//Load arbiter with beam parameter sets
AssertTrue(fbArbiter.AddRequest(nEVReqID, stEVReqBP, sDevName:= 'Device'),
                    'Safest stEVReqBP request failed to load');

//Load arbiter with beam parameter sets
AssertTrue(fbArbiter.AddRequest(nRateReqID, stRateReqBP, sDevName:= 'Device'),
                    'Safest stRateReqBP request failed to load');

//Load arbiter with beam parameter sets
AssertTrue(fbArbiter.AddRequest(nBCRangeReqID, stBCReqBP, sDevName:= 'Device'),
                    'Safest stBCReqBP request failed to load');

stArbitratedBP := fbArbiter.GetArbitratedBP();

AssertFalse(F_DifferentBeamParams(stExpectedBP, stArbitratedBP),
                'Arbitrated BP does not match expected.');

TEST_FINISHED();
END_METHOD

METHOD DoS
VAR



    nOrigReqID : UDINT := 30;
    nSecondReqID : UDINT := 35;

    nPeskyReqID : UDINT := 40;


END_VAR
VAR_INST
    DosArb : FB_Arbiter(20);

    DummyHA : FB_DummyHA := (ReqAcknowledged:=FALSE); // Set req ack false to start so we can control when it is verified
    nTimeoutCounter : UINT;
    bInit : BOOL;
    bSecond : BOOL;
    eDosTestCases : E_ArbDosTestStates;
END_VAR
VAR CONSTANT
        nTimeoutCounterMAX : UINT := 50;
        nWaitCount : UINT := 10;
        nWait2ndCount : UINT := nWaitCount + 5;
END_VAR
TEST('DoS');

CASE eDosTestCases OF
    E_ArbDosTestStates.Init: // Init, first request
        DosArb.AddRequest(nOrigReqID, PMPS_GVL.cst0RateBeam, sDevName:= 'Device');
        eDosTestCases := E_ArbDosTestStates.SecondReq;

    E_ArbDosTestStates.SecondReq: // Add second request
        DosArb.AddRequest(nSecondReqID, PMPS_GVL.cst0RateBeam, sDevName:= 'Device');
        eDosTestCases := E_ArbDosTestStates.WaitForAck;

    E_ArbDosTestStates.WaitForAck:
        IF nTimeoutCounter > nWaitCount THEN
            DummyHA.ReqAcknowledged := TRUE;
            eDosTestCases := E_ArbDosTestStates.WaitFor2ndAck;
        END_IF

    E_ArbDosTestStates.WaitFor2ndAck:
        DummyHA.ReqAcknowledged := False;
        IF nTimeoutCounter > nWait2ndCount THEN
            DummyHA.ReqAcknowledged := TRUE;
            eDosTestCases := E_ArbDosTestStates.RunAsserts;
        END_IF

END_CASE

DosArb.ElevateRequest(DummyHA);

// Pesky request always adding and removing
DosArb.RemoveRequest(nPeskyReqID);
DosArb.AddRequest(nPeskyReqID, PMPS_GVL.cst0RateBeam, sDevName:= 'Device');


nTimeoutCounter := nTimeoutCounter + 1;

IF nTimeoutCounter > nTimeoutCounterMAX or eDosTestCases = E_ArbDosTestStates.RunAsserts THEN
    AssertTrue(DosArb.CheckRequest(nOrigReqID), 'Original request still not accepted');
    AssertTrue(DosArb.CheckRequest(nSecondReqID), 'Second request still not accepted');

    TEST_FINISHED_NAMED('DoS');
END_IF
END_METHOD

{attribute 'no_check'}
METHOD FullArbitrationStack
VAR_INPUT
END_VAR
VAR
    nId    :    DWORD := 1;
    stReq    :    ST_BeamParams := (nTran:=12);

    nIdDoS : DWORD := 13;
    stDoSReq : ST_BeamParams := PMPS_GVL.cstFullBeam;
END_VAR
VAR_INST
    fbArbiter    :    FB_Arbiter(1);

    fbHigherArb : FB_Arbiter(2);

    fbSubSysToArb : FB_SubSysToArbiter_IO; // Subsystem interface with beamline arbiter PLC
    pBPR : POINTER TO ST_BeamParams_IO;

    fbArbToSubSys : FB_ArbiterToSubSys_IO := (RequestingSystemID:=42); // Beamline arbiter PLC interface with subsystems
    pBPC : POINTER TO ST_BeamParams_IO;

    fbBPR : FB_BPRequestor; // Use in the arbiter PLC to apply an arbitrated beam parameter set to the accelerator interface

    FFO : FB_HardwareFFOutput; // Dummy FFO not important for these tests

    Cycle : INT := 0;

    CycleLimit : INT := 20;

END_VAR
VAR CONSTANT
    SysID : DWORD := 42;
END_VAR
// This simulates a synchronous cycle between the subsystem and arbiter PLC cycles. Ie. phase is locked, and cycle time is the same. This is not always the case, so these tests should be
// trusted with a grain of salt.

TEST('FullStack');



CASE Cycle OF

0:
    IF NOT fbArbiter.CheckRequestInPool(nID) THEN
        AssertTrue(fbArbiter.AddRequest(nId, stReq,'Device'), 'Arbiter returned false from AddRequest'); // some device asking its local arbiter for some beam parameters
    END_IF

    TEST('JustEnteredRequest');
    AssertFalse(fbArbiter.CheckRequest(nId),
        'Check should fail. Request not arbitrated yet.');
    TEST_FINISHED();

8000:
    TEST_FINISHED_NAMED('FullStack');

END_CASE


TEST('VerifyBPRHasBP');
IF fbHigherArb.CheckRequest(SysID) THEN
    AssertFalse(F_DifferentBeamParams(stReq, fbBPR.q_ReqBP),
        'Beam parameters not fully propagated to BPR at highest level');
        TEST_FINISHED_NAMED('VerifyBPRHasBP');
END_IF

TEST('ArbToSubsysPropagation');
IF fbArbToSubSys.nActiveCohort = fbArbToSubSys.nRequestedCohort
    AND fbArbToSubSys.nActiveCohort <> 0 THEN
    AssertTrue(fbHigherArb.CheckRequest(SysID),
        'Active cohort = Requested cohort before higher arbiter confirmed request was active');
    TEST_FINISHED_NAMED('ArbToSubsysPropagation');
END_IF

TEST('SubsysToArbPropagation');
IF fbArbiter.CheckRequest(nId) THEN
    AssertTrue(fbSubSysToArb.nActiveCohort >= fbSubSysToArb.nRequestCohort,
        'Request validated before higher level confirmation');
    TEST_FINISHED_NAMED('SubsysToArbPropagation');
END_IF


TEST('VerifyIncludedAtAllLevels');
IF fbArbiter.CheckRequest(nId) THEN
    AssertTrue(fbHigherArb.CheckRequest(fbArbToSubSys.RequestingSystemID), 'HigherArb is not yet included in arbitration');
    AssertTrue(fbSubSysToArb.CheckRequest(fbArbiter.nLowerAuthorityID), 'Local Arb is not yet included in arbitration');
    TEST_FINISHED_NAMED('VerifyIncludedAtAllLevels');
END_IF


///////////////////////////////////////
//Sub system cycle
fbSubSysToArb(Arbiter := fbArbiter, fbFFHWO := FFO);
//END of sub system cycle
///////////////////////////////////////

//Ethercat transfer simulation
// Transfer of requested BP to arbiter PLC
pBPR := ADR(fbArbToSubSys.i_RequestedBP);
pBPR^ := fbSubSysToArb.q_stRequestedBP;

// Transfer of current BP to sub system PLC
pBPC := ADR(fbSubSysToArb.i_stCurrentBP);
pBPC^ := fbArbToSubSys.o_CurrentBP;

//////////////////////////////////////
//Start of arbiter plc cycle
//Arb io collects sub system status
fbArbToSubSys(Arbiter := fbHigherArb, fbFFHWO := FFO); // This is making a request in the higher arb
//BPR collects arbiter summation
fbBPR(Arbiter := fbHigherArb); // This is getting the arbitrated BP




IF CycleLimit > Cycle THEN
    Cycle := Cycle + 1;
ELSE
    Cycle := 8000;
END_IF
END_METHOD

METHOD RemoveReq
VAR

    Arb : FB_Arbiter(20);

    DummyHA : FB_DummyHA;

    Result : BOOL;

END_VAR

Arb.AddRequest(30, PMPS_GVL.cst0RateBeam, 'Device');

Arb.ElevateRequest(DummyHA);

TEST('Remove Req');
    Result := Arb.RemoveRequest(77);

    AssertFalse( Result, 'RemoveReq returned true, with nothing to remove');
    AssertFalse( Arb.bStartNewAckRequest , 'StartNewAckRequest is set. Something is wrong');

TEST_FINISHED();
END_METHOD

METHOD RequestCheckRemoveBP
VAR_INPUT
END_VAR
VAR

    nId    :    DWORD := 1;
    stReq    :    ST_BeamParams;
END_VAR
VAR_INST
    fbArbiter    :    FB_Arbiter(1);
END_VAR
TEST('RequestBP');
AssertTrue(fbArbiter.AddRequest(nId, stReq, 'Device'),
    'Request failed');

TEST_FINISHED();

TEST('DuplicateID');
AssertFalse(fbArbiter.AddRequest(nId, stReq, 'Device'),
    'Duplicate request accepted, not good.');

TEST_FINISHED();

TEST('CheckBP');
AssertFalse(fbArbiter.CheckRequest(nId),
    'Check should fail. Request not arbitrated yet.');
TEST_FINISHED();

TEST('CheckBPArbitrated');
WRITE_PROTECTED_ULINT(ADR(fbArbiter.nActiveCohort), fbArbiter.nNextCohort);
AssertTrue(fbArbiter.CheckRequest(nId),
    'Check should pass.');

TEST_FINISHED();

TEST('IDDoesNotExist');

AssertFalse(fbArbiter.CheckRequest(nId+1),
    'Check returned true when ID does not exist');

TEST_FINISHED();

TEST('RemoveBP');
AssertTrue(fbArbiter.RemoveRequest(nId),
    'Remove failed');
AssertFalse(fbArbiter.CheckRequest(nId),
    'Remove did not remove request');

TEST_FINISHED();

TEST('NoRequestsFullBeam');

AssertFalse(F_DifferentBeamParams(fbArbiter.GetArbitratedBP(), PMPS_GVL.cstFullBeam), 'Arbitrated beam should be full with all requests removed');

TEST_FINISHED();
END_METHOD

METHOD StackArbiters
VAR_INPUT
END_VAR
VAR
    nId    :    DWORD := 1;
    stReq    :    ST_BeamParams := (nTran:=12);
END_VAR
VAR_INST
    fbArbiter    :    FB_Arbiter(1);

    fbHigherArb : FB_Arbiter(2);

    ArbBP : ST_BeamParams;

    Cycle : INT := 0;

    CycleLimit : INT := 20;

END_VAR
VAR CONSTANT
    SysID : DWORD := 42;
END_VAR

TEST('StackingArbiters');
fbArbiter.AddRequest(nReqID:=nId, stReqBP:=stReq, sDevName :='Device');

fbArbiter.ElevateRequest(fbHigherArb);

ArbBP := fbHigherArb.GetArbitratedBP();

AssertTrue(ArbBP.nTran = 12, 'We should see the transmission number here');

TEST_FINISHED();
END_METHOD

END_FUNCTION_BLOCK

// TestComponents/FB_ArbToSubsys_Test
{attribute 'call_after_init'}
FUNCTION_BLOCK FB_ArbToSubsys_Test EXTENDS TcUnit.FB_TestSuite
VAR_INPUT
END_VAR
VAR_OUTPUT
END_VAR
VAR
END_VAR

BasicFunction();

{attribute 'no_check'}
METHOD BasicFunction
VAR_INPUT
END_VAR
VAR CONSTANT
    SysID : DWORD := 42;
END_VAR
VAR
    nId    :    DWORD := 1;
    stReq    :    ST_BeamParams := (nTran:=12);
END_VAR
VAR_INST
    fbArbiter    :    FB_Arbiter(1);

    pBPR : POINTER TO ST_BeamParams_IO;

    stBPRIO : ST_BeamParams_IO := (
        nCohortInt := 1,
        nTran := 35); // Simulates subsystem BP request

    fbArbToSubSys : FB_ArbiterToSubSys_IO := (RequestingSystemID:=42); // Beamline arbiter PLC interface with subsystems
    pBPC : POINTER TO ST_BeamParams_IO;

    fbBPR : FB_BPRequestor; // Use in the arbiter PLC to apply an arbitrated beam parameter set to the accelerator interface

    FFO : FB_HardwareFFOutput; // Dummy FFO not important for these tests

    Cycle : INT := 0;

    CycleLimit : INT := 20;

END_VAR

// Simulate an initial cycle with no new requests coming in
fbBPR(Arbiter:=fbArbiter);
fbArbToSubSys(Arbiter:=fbArbiter, fbFFHWO:=FFO);

TEST('Init');
TEST_FINISHED();

//Ethercat transfer simulation
// Transfer of requested BP to arbiter PLC
pBPR := ADR(fbArbToSubSys.i_RequestedBP);
pBPR^ := stBPRIO;

///////////////////////////////////////
//Sub system cycle
fbBPR(Arbiter:=fbArbiter);
fbArbToSubSys(Arbiter:=fbArbiter, fbFFHWO:=FFO);
//END of sub system cycle
///////////////////////////////////////


TEST('New request');
    AssertTrue(fbArbToSubSys.nRequestedCohort = fbArbToSubSys.i_RequestedBP.nCohortInt, 'ReqCohort and qBP Cohort do not match, and they should');
    AssertTrue(fbArbiter.CheckRequestInPool(SysID), 'ArbToSubSys request should be in arbiter pool now');
    AssertTrue(fbArbToSubSys.nActiveCohort = 0, 'Active cohort should remain the initial value until the current request is active in higher arbitration');
    AssertTrue(fbArbToSubSys.o_CurrentBP.nCohortInt = fbArbToSubSys.nActiveCohort, 'Cohort being sent to sub system remains unincremented');
TEST_FINISHED_NAMED('New request');


///////////////////////////////////////
//Sub system cycle
fbBPR(Arbiter:=fbArbiter);
fbArbToSubSys(Arbiter:=fbArbiter, fbFFHWO:=FFO);
//END of sub system cycle
///////////////////////////////////////

///////////////////////////////////////
//Sub system cycle
fbBPR(Arbiter:=fbArbiter);
fbArbToSubSys(Arbiter:=fbArbiter, fbFFHWO:=FFO);
//END of sub system cycle
///////////////////////////////////////

///////////////////////////////////////
//Sub system cycle
fbBPR(Arbiter:=fbArbiter);
fbArbToSubSys(Arbiter:=fbArbiter, fbFFHWO:=FFO);
//END of sub system cycle
///////////////////////////////////////

TEST('Request has become active');
    AssertTrue(fbArbToSubSys.nRequestedCohort = fbArbToSubSys.nActiveCohort, 'ReqCohort and qBP Cohort do not match, and they should');
    AssertTrue(fbArbiter.CheckRequest(SysID), 'ArbToSubSys request should be in arbiter pool now');
    AssertTrue(fbArbToSubSys.nActiveCohort = stBPRIO.nCohortInt, 'Active cohort should remain the initial value until the current request is active in higher arbitration');
    AssertTrue(fbBPR.q_ReqBP.nTran = stBPRIO.nTran, 'BPR and requested BP should match');
TEST_FINISHED_NAMED('Request has become active');
END_METHOD

END_FUNCTION_BLOCK

// TestComponents/FB_AttenuatorSimulator
FUNCTION_BLOCK FB_AttenuatorSimulator
VAR_INPUT
    i_rRequestedAttenuation    :    REAL;
    i_stBPReadback    :    ST_BeamParams;
END_VAR
VAR_OUTPUT
    q_xFault    :    BOOL;
    q_rCurrentAttenuation    :    REAL;
END_VAR
VAR_IN_OUT
    Arbiter    :    FB_Arbiter; //Higher level arbiter from which upstream attenuation can be requested
END_VAR
VAR
    tonDelay    :    TON := (
        PT := T#3S
        );
END_VAR

// Really basic delay
tonDelay(IN := i_rRequestedAttenuation <> q_rCurrentAttenuation);

IF tonDelay.Q THEN
    q_rCurrentAttenuation := i_rRequestedAttenuation;
END_IF

END_FUNCTION_BLOCK

// TestComponents/FB_BPTM_Test
{attribute 'call_after_init'}
FUNCTION_BLOCK FB_BPTM_Test EXTENDS TcUnit.FB_TestSuite
VAR_INPUT
END_VAR
VAR_OUTPUT
END_VAR
VAR
END_VAR
VAR CONSTANT
    BPTM_ARR : UDINT := PMPS_PARAM.MAX_ASSERTIONS;
    cCycle : UINT := 20; // How many cycles does it take to complete a BPTM
END_VAR

BPTMBasicFunction();
InterruptAtAllSteps();
FullArbError();

METHOD BPTMBasicFunction
VAR_INPUT
END_VAR
VAR
    //Final and transition assertions
    nTransitionID    :    UDINT := 1;
    stTransitionAssertion    :    ST_BeamParams := (nRate := 10, nBCRange:=0);

    nReqID    :    UDINT    := 2;
    stReqAssertion    :    ST_BeamParams := (nTran := 0.2, nBCRange:=2#0000_0000_0000_0011);

END_VAR
VAR_INST
    fbBPTM_TestBasicFunction    :    BeamParameterTransitionManager;
    fbArbiter    :    FB_Arbiter(1);
    ffo : FB_HardwareFFOutput;
    fbSubSysIO : FB_DummyArbIO;
    xFirstPass    :    BOOL := TRUE;
    eTestStep: E_BPTMTestStates := E_BPTMTestStates.Init;
END_VAR

// Completes arbiter request elevation process
// Necessary for CheckRequest to return true, ever
    fbBPTM_TestBasicFunction(
        fbArbiter := fbArbiter,
        );

fbSubSysIO(LA := fbArbiter, FFO := ffo);

// Note: this struct may also be (over)written to in the tests below, specifically rate.
fbBPTM_TestBasicFunction.stCurrentBeamParameters := fbSubSysIO.q_stSimulatedBPReadback;

//MG: Need to set the Machine mode testing SC
PMPS_GVL.stCurrentBeamParameters.nMachineMode :=0;

CASE eTestStep OF

E_BPTMTestStates.Init:

    TEST('BPTMTest');
    eTestStep := E_BPTMTestStates.WaitingForBeam;

E_BPTMTestStates.WaitingForBeam:
    TEST('BPTM Waits for Beam');

    fbBPTM_TestBasicFunction.i_TransitionAssertionID := nTransitionID;
    fbBPTM_TestBasicFunction.i_stTransitionAssertion := stTransitionAssertion;

    fbBPTM_TestBasicFunction.i_nRequestedAssertionID := nReqID;
    fbBPTM_TestBasicFunction.i_stRequestedAssertion := stReqAssertion;

    IF fbBPTM_TestBasicFunction.eBPTMState = E_BPTMState.WaitForBP AND
        NOT fbBPTM_TestBasicFunction.xEntry THEN

        AssertTrue(fbArbiter.CheckRequestInPool(nTransitionID), 'Arbiter did not accept BPTM transition assertion');

        AssertTrue(fbArbiter.CheckRequestInPool(nReqID), 'Arbiter did not accept BPTM transition assertion');

        AssertFalse(fbBPTM_TestBasicFunction.q_xTransitionAuthorized,
            'Transition should not be authorized until requests are in and beam is ready');

        AssertTrue(fbBPTM_TestBasicFunction.bBusy, 'Busy should be true here');
        AssertFalse(fbBPTM_TestBasicFunction.bDone, 'Done should be false');
        AssertFalse(fbBPTM_TestBasicFunction.bError, 'Error should be false here');

        TEST_FINISHED_NAMED('BPTM Waits for Beam');

        eTestStep := E_BPTMTestStates.Transitioning;
    END_IF


E_BPTMTestStates.Transitioning:
    TEST('BPTM Authorizes Transition');

    fbBPTM_TestBasicFunction.stCurrentBeamParameters.nRate := 0; // satisfies the transition request
    fbBPTM_TestBasicFunction.stCurrentBeamParameters.nBeamClass := 0; // satisfies the transition request

    IF fbBPTM_TestBasicFunction.eBPTMState = E_BPTMState.Transitioning AND
        NOT fbBPTM_TestBasicFunction.xEntry THEN

        AssertTrue(fbArbiter.CheckRequest(nTransitionID),
            'Transition assertion should be in arbiter');

        AssertTrue(fbArbiter.CheckRequest(nReqID),
            'Final assertion should be in arbiter');

        AssertTrue(fbBPTM_TestBasicFunction.q_xTransitionAuthorized,
            'Transition should be authorized at this point.');

        AssertEquals(nReqID, fbBPTM_TestBasicFunction.nCurrentAssertionID,
            'nCurrentAssertionID not set.');

        TEST_FINISHED_NAMED('BPTM Authorizes Transition');

        eTestStep := E_BPTMTestStates.WaitingForFinalAssertion;
    END_IF

E_BPTMTestStates.WaitingForFinalAssertion:
    TEST('BPTM Waits for final BP');

    fbBPTM_TestBasicFunction.i_xDoneMoving := TRUE;

    IF fbBPTM_TestBasicFunction.eBPTMState = E_BPTMState.WaitForFinalBP THEN

        AssertTrue(fbArbiter.CheckRequest(nTransitionID),
        'Transition assertion should be in arbiter');

        TEST_FINISHED_NAMED('BPTM Waits for final BP');

        eTestStep := E_BPTMTestStates.CleaningUp;
    END_IF

E_BPTMTestStates.CleaningUp:

    fbSubSysIO.AutoUpdateBP := TRUE;

    TEST('Cleaning up');

    IF fbBPTM_TestBasicFunction.eBPTMState = E_BPTMState.Done THEN

        AssertFalse(fbArbiter.CheckRequestInPool(nTransitionID), 'Transition req should be removed from arb now');

        eTestStep := E_BPTMTestStates.Done;

        TEST_FINISHED_NAMED('Cleaning up');
    END_IF

E_BPTMTestStates.Done:


    AssertTrue(fbBPTM_TestBasicFunction.bDone, 'Done should be set');
    AssertFalse(fbBPTM_TestBasicFunction.bError, 'Error should be cleared');
    AssertFalse(fbBPTM_TestBasicFunction.bBusy, 'Busy should be false');

    TEST_FINISHED_NAMED('BPTMTest');

END_CASE
END_METHOD

// Simulate error due to full arbiter
METHOD FullArbError
VAR_INPUT
END_VAR
VAR
    //Final and transition assertions
    nTransitionID    :    UDINT := 1000;
    stTransitionAssertion    :    ST_BeamParams :=  ( nTran := 0, neVRange := 0, nRate  := 0);//PMPS_GVL.cstSafeBeam;

    nReqID    :    UDINT    := 2000;
    stReqAssertion    :    ST_BeamParams := ( nTran := 0, neVRange := 0, nRate  := 0);//PMPS_GVL.cstSafeBeam;

    idx : UDINT;

    nRandID : DWORD;
    testReq : ST_BeamParams := (neVRange := 16#FFEE, nRate:=33);

END_VAR
VAR_INST
    fbBPTM_TestFullArb    :    BeamParameterTransitionManager;
    fbArbFullErr    :    FB_Arbiter(1);
    ffo : FB_HardwareFFOutput;
    fbSubSysIO : FB_DummyArbIO;
    fbBPR :  FB_BPRequestor;
    xFirstPass    :    BOOL := TRUE;
    eTestStep: E_BPTMTestStates := E_BPTMTestStates.Init;
    tonRetryTimeout : TON := (PT:=T#5s);
    entryToRetry : bool := true;
    fbRand : DRAND := (Seed :=1);
END_VAR
CASE eTestStep OF

E_BPTMTestStates.Init:

    TEST('BPTMErrorFullArb');

    // Fill the arbiter
    FOR idx := 1 TO PMPS_PARAM.MAX_ASSERTIONS // this fills the arbiter
                    - fbBPTM_TestFullArb.cReqArbCapacity + 1 DO // but test just one over the allowed amount
        fbArbFullErr.AddRequest(nReqID := idx, stReqBP := testReq, sDevName :='Device');
    END_FOR

    fbSubSysIO.AutoUpdateBP := TRUE;

    AssertTrue(PMPS_PARAM.MAX_ASSERTIONS - fbArbFullErr.nEntryCount < fbBPTM_TestFullArb.cReqArbCapacity,
        'Arbiter is not full enough, rest of tests will be invalid');

    eTestStep := E_BPTMTestStates.Error;

E_BPTMTestStates.Error:

    TEST('BPTM Full Error');

    IF fbBPTM_TestFullArb.bError THEN

        AssertTrue(fbBPTM_TestFullArb.bError AND fbBPTM_TestFullArb.nErrId = PMPS_CODES.NoRoomInArb,
            'Incorrect error response from full arbiter.');

        TEST_FINISHED_NAMED('BPTM Full Error');

        eTestStep := E_BPTMTestStates.Retry;

    END_IF

E_BPTMTestStates.Retry:

    TEST('Test Retry Post Failed Final');

    // Clear the arbiter
    if entryToRetry THEN
        FOR idx := 1 TO PMPS_PARAM.MAX_ASSERTIONS + 1 DO
            fbArbFullErr.RemoveRequest(idx);
        END_FOR
        entryToRetry := FALSE;
    END_IF

    // Push the retry button
    fbBPTM_TestFullArb.bRetry := TRUE;

    tonRetryTimeout(IN:=TRUE);

    IF tonRetryTimeout.Q OR fbBPTM_TestFullArb.q_xTransitionAuthorized THEN
        AssertTrue(fbBPTM_TestFullArb.q_xTransitionAuthorized, 'Transition should have been authorized by now');
        AssertTrue(fbArbFullErr.CheckRequest(nTransitionID), 'Transition ID is missing from arbiter while transition is authorized');
        AssertTrue(fbArbFullErr.CheckRequest(nReqID), 'Final ID is missing from arbiter while transition is authorized');

        TEST_FINISHED_NAMED('Test Retry Post Failed Final');

        eTestStep := E_BPTMTestStates.CleaningUp;
    END_IF

E_BPTMTestStates.CleaningUp:
    TEST_FINISHED_NAMED('BPTMErrorFullArb');

END_CASE

fbBPTM_TestFullArb(
    fbArbiter := fbArbFullErr,
    i_TransitionAssertionID := nTransitionID,
    i_stTransitionAssertion := stTransitionAssertion,

    i_nRequestedAssertionID := nReqID,
    i_stRequestedAssertion := stReqAssertion,

    stCurrentBeamParameters := fbSubSysIO.q_stSimulatedBPReadback,
);

fbSubSysIO(LA := fbArbFullErr, FFO := ffo);
END_METHOD

// Test the BPTM seamlessly handles new requests at any stage
// Verify old requests are removed from arbiter
{attribute 'no_check'}
METHOD InterruptAtAllSteps
VAR_INPUT
END_VAR
VAR
    //Final and transition assertions
    nTransitionID    :    UDINT := 16#DAAD;
    stTranReq    :    ST_BeamParams := PMPS_GVL.cst0RateBeam;

    nFirstReqID    :    UDINT    := 16#FEED;
    stFirstReq    :    ST_BeamParams := (nTran :=1, nRate := 16#FEED, neVRange :=2#1111_1111_1111_1111_1111_1111_1111_1111);

END_VAR
VAR_INST
    fbBPTM_InterruptionTest    :    BeamParameterTransitionManager;

    ffo : FB_HardwareFFOutput := (bAutoReset:=TRUE);
    fbSubSysIO : FB_DummyArbIO;
    fbBPR :  FB_BPRequestor;
    xFirstPass    :    BOOL := TRUE;
    eTestStep: E_BPTMTestStates := E_BPTMTestStates.Init;
    tonRetryTimeout : TON := (PT:=T#5s);

    fbBPTMDiscCycles : BeamParameterTransitionManager;
    fbSubSysIODisc : FB_DummyArbIO;
    fbArbDisc : FB_Arbiter(1000);

    iCount : UINT;

    aBPTM : ARRAY [1..cCycle] OF BeamParameterTransitionManager;
    BPTMUnderTest : REFERENCE TO BeamParameterTransitionManager;
    fbArbiter    :    FB_Arbiter(1);
    aArbIO : ARRAY [1..cCycle] OF FB_DummyArbIO;
    ArbIO : REFERENCE TO FB_DummyArbIO;
    nCycleLim : UINT;
    nCycle : UINT;
    sCurrentTestName : STRING :='';
    bCycleLimHit : BOOL;
    nAllStepsDone : BYTE;
    tTimeOut : TON := (PT:=T#20ms);

    bTestedOnce : BOOl;
END_VAR
VAR CONSTANT
    nNewTarget : INT := 0;
    nRequestBP : INT := 1;
    nWaitForBP : INT := 2;
    nTransitioning : INT := 3;
    nWaitForFinalBP : INT := 4;
    nCleaningUp : INT := 5;
    nDone : INT := 6;
    nIdle : INT := 7;
END_VAR

(* These tests will confirm the BPTM is interruptable at any step,
meaning it will not deadlock or stall, and will always complete with
the correct sequencing *)

(* This functionality is crucial as a deadlocked BPTM will need manual intervention,
users of the BPTM should always be able to just set a target BP that is easy to reach
at any point in time, and have the BPTM head in that direction and succeed. *)

// Determine how many cycles it would take normally, to complete a full BPTM cycle
// This count will be verified against the current count constant

IF NOT bTestedOnce THEN

TEST('CheckBPTM Cycle Count');

WHILE fbBPTMDiscCycles.eBPTMState <> E_BPTMState.Idle DO

    fbBPTMDiscCycles.i_TransitionAssertionID := nTransitionID;
    fbBPTMDiscCycles.i_stTransitionAssertion := stTranReq;

    fbBPTMDiscCycles.i_nRequestedAssertionID := nFirstReqID;
    fbBPTMDiscCycles.i_stRequestedAssertion := stFirstReq;

    fbBPTMDiscCycles(fbArbiter:=fbArbDisc);
    fbSubSysIODisc(LA:=fbArbDisc, FFO:=ffo);

    fbBPTMDiscCycles.stCurrentBeamParameters := fbSubSysIODisc.q_stSimulatedBPReadback;

    fbSubSysIODisc.AutoUpdateBP := TRUE;

    fbBPTMDiscCycles.i_xDoneMoving S= fbBPTMDiscCycles.q_xTransitionAuthorized;

    iCount := iCount + 1;
END_WHILE

IF fbBPTMDiscCycles.eBPTMState = E_BPTMState.Idle THEN
    AssertTrue(cCycle >= iCount, CONCAT('cCycle is too low, increase it to', INT_TO_STRING(iCount)));
    TEST_FINISHED_NAMED('CheckBPTM Cycle Count');
END_IF

// Run BPTM for nCycleLim cycles, switch to a new target, verify BPTM completes anyways

FOR nCycleLim := 1 TO cCycle DO

    nCycle := 0;

    bCycleLimHit := FALSE;

    BPTMUnderTest REF= aBPTM[nCycleLim];
    ArbIO REF= aArbIO[nCycleLim];

    BPTMUnderTest.i_TransitionAssertionID := nTransitionID;
    BPTMUnderTest.i_stTransitionAssertion := stTranReq;

    ArbIO.AutoUpdateBP := TRUE;

    // Start the test for this Cycle Limit
    sCurrentTestName := CONCAT('CycleLimTest:',INT_TO_STRING(nCycleLim));
    TEST(sCurrentTestName);

    nAllStepsDone := 0;

    tTimeOut(IN:=FALSE);

    WHILE nAllStepsDone <> 16#FF DO

        tTimeOut(IN:= TRUE);

        IF tTimeOut.Q THEN
            AssertTrue(FALSE, CONCAT('Failed ', BYTE_TO_HEXSTR(nAllStepsDone, 2, FALSE)));
            EXIT;
        END_IF

        // Verify all steps complete
        IF bCycleLimHit THEN
            nAllStepsDone.nNewTarget S= BPTMUnderTest.eBPTMState = E_BPTMState.NewTarget;
            nAllStepsDone.nRequestBP S= BPTMUnderTest.eBPTMState = E_BPTMState.RequestBP;
            nAllStepsDone.nWaitForBP S= BPTMUnderTest.eBPTMState = E_BPTMState.WaitForBP;
            nAllStepsDone.nTransitioning S= BPTMUnderTest.eBPTMState = E_BPTMState.Transitioning;
            nAllStepsDone.nWaitForFinalBP S= BPTMUnderTest.eBPTMState = E_BPTMState.WaitForFinalBP;
            nAllStepsDone.nCleaningUp S= BPTMUnderTest.eBPTMState = E_BPTMState.CleaningUp;
            nAllStepsDone.nDone S= BPTMUnderTest.eBPTMState = E_BPTMState.Done;
            nAllStepsDone.nIdle S= BPTMUnderTest.eBPTMState = E_BPTMState.Idle;
        ELSE
            nAllStepsDone := 0;
        END_IF

        // After nCycleLim cycles (nCycle), change the target
        IF nCycle >= nCycleLim THEN
            BPTMUnderTest.i_nRequestedAssertionID := nCycleLim;
            BPTMUnderTest.i_stRequestedAssertion.nRate := nCycleLim;
            bCycleLimHit := TRUE;
        ELSE
            BPTMUnderTest.i_nRequestedAssertionID := nFirstReqID;
            BPTMUnderTest.i_stRequestedAssertion := stFirstReq;
        END_IF

        BPTMUnderTest(fbArbiter:=fbArbiter);
        ArbIO(LA:=fbArbiter, FFO := ffo);

        BPTMUnderTest.stCurrentBeamParameters := ArbIO.q_stSimulatedBPReadback;

        BPTMUnderTest.i_xDoneMoving := BPTMUnderTest.q_xTransitionAuthorized;

        nCycle := nCycle + 1;

    END_WHILE

    AssertTrue(fbArbiter.CheckRequestInPool(BPTMUnderTest.i_nRequestedAssertionID),
        CONCAT('Final req not in pool: ', UINT_TO_STRING(nCycleLim)));
    AssertFalse(fbArbiter.CheckRequestInPool(BPTMUnderTest.i_TransitionAssertionID),
        'TransReq still in pool');
    AssertFalse(fbArbiter.CheckRequestInPool(nFirstReqID),
        'First req still in pool');
    AssertTrue(bCycleLimHit,
        CONCAT('Cycle lim not hit', UINT_TO_STRING(nCycleLim)));
    AssertTrue(ArbIO.q_stSimulatedBPReadback.nRate = BPTMUnderTest.i_stRequestedAssertion.nRate,
        'Rates are not equal...');

    TEST_FINISHED_NAMED(sCurrentTestName);

    // Clean up for next test

    fbArbiter.RemoveRequest(nFirstReqID);
    fbArbiter.RemoveRequest(nTransitionID);
    fbArbiter.RemoveRequest(nCycleLim);

END_FOR

END_IF
END_METHOD

END_FUNCTION_BLOCK

// TestComponents/FB_DiffBP_Test
{attribute 'call_after_init'}
FUNCTION_BLOCK FB_DiffBP_Test EXTENDS TcUnit.FB_TestSuite
VAR_INPUT
END_VAR
VAR_OUTPUT
END_VAR
VAR

END_VAR


BPDiff();

//Verify BP comparison remains logical.
METHOD BPDiff
VAR_INPUT
END_VAR
VAR
    BP1    :    ST_BeamParams;
    BP2    :    ST_BeamParams;
END_VAR
TEST('BPDiffCheck');

BP2.nTran := 10;

AssertTrue(
    F_DifferentBeamParams(BP1, BP2),
    'DifferentBP eval is broken (True)');

BP1.nTran := BP2.nTran;

AssertFalse(
    F_DifferentBeamParams(BP2, BP1),
    'DifferentBP eval is broken (False)');

TEST_FINISHED();
END_METHOD

END_FUNCTION_BLOCK

// TestComponents/FB_evRangeCalculator_Test
{attribute 'call_after_init'}
FUNCTION_BLOCK FB_evRangeCalculator_Test EXTENDS FB_TestSuite
VAR_INPUT
END_VAR
VAR_OUTPUT
END_VAR
VAR
END_VAR
VAR CONSTANT
    RandomBoundary : INT := 2;
END_VAR

BasicFunction();

{attribute 'no_check'}
METHOD BasicFunction
VAR_INPUT
END_VAR
VAR
    {attribute 'displaymode' := 'binary'}
    LastWord : DWORD := 2#0000_0000_0000_0000_0000_0000_0000_0010;
    {attribute 'displaymode' := 'binary'}
    Result : DWORD;
    {attribute 'displaymode' := 'binary'}
    TestEV : DWORD;

    {attribute 'displaymode' := 'binary'}
    tEvW : DWORD;
    tEv : REAL;


    fbStr : FB_FormatString;

    MiscNumber : INT;
END_VAR
VAR CONSTANT
    nLowerLimitBoundary : INT := 0;

    RandomBoundary : INT := 2;
    MNU : INT := 3; //RandomBoundary + 1
    MND : INT := 1; //RandomBoundary - 1
END_VAR
Test('CheckRanges');

//Lower limit equal
tEvW.nLowerLimitBoundary := TRUE;
tEv := PMPS_GVL.g_areVBoundaries[nLowerLimitBoundary];
Result := F_eVRangeCalculator(tEv, 0);
AssertTrue(
    Result = tEvW,
    'Lower limit not inclusive');

// Lower range flags
tEvW.nLowerLimitBoundary := TRUE;
tEv := PMPS_GVL.g_areVBoundaries[nLowerLimitBoundary] / 2;
Result := F_eVRangeCalculator(tEv, 0);
AssertTrue(
    Result = tEvW,
    'eV below lower range should come back true');

//Mid range
tEvW := 0;
tEvW.RandomBoundary := TRUE;
//ev result that is smack dab in the middle of a range
tEv := PMPS_GVL.g_areVBoundaries[RandomBoundary] - ((PMPS_GVL.g_areVBoundaries[RandomBoundary] - PMPS_GVL.g_areVBoundaries[MND]) / 2);
Result := F_eVRangeCalculator(tEv, 0);
AssertTrue(
    Result = tEvW,
    'In range failed, whatever you did, it broke this really bad.');

//Out of range
tEvW := 0;
tEvW.RandomBoundary := TRUE;
//Ev result that is beyond the current range (midway into the next range up)
tEv := PMPS_GVL.g_areVBoundaries[MNU] - (PMPS_GVL.g_areVBoundaries[MNU]-PMPS_GVL.g_areVBoundaries[RandomBoundary])/2;
Result := F_eVRangeCalculator(tEv, 0);
AssertFalse(
    Result = tEvW,
    'Out of range failed, whatever you did, it broke this really bad.');

TEST_FINISHED();

Test('Negative eV failsafes');
//Negative eV
AssertTrue(
    F_eVRangeCalculator(-300, 0) = 16#FFFF_FFFF,
    'Working with antimatter? Negative eV should failsafe to FFFF.');

TEST_FINISHED();

Test('Out of range eV failsafes');
// eV too high
AssertTrue(
    F_eVRangeCalculator(PMPS_GVL.g_areVBoundaries[PMPS_GVL.g_cBoundaries] + 1, 0) = 16#FFFF_FFFF,
    'eV above the last threshold should failsafe.');

TEST_FINISHED();

Test('Check hyst keeps');

LastWord := F_eVRangeCalculator(PMPS_GVL.g_areVBoundaries[RandomBoundary], 2#0000_0000_0000_0000_0000_0000_0000_0000);

// Last word should be 2#0000_0000_0000_0100

    Result := F_eVRangeCalculator(
        PMPS_GVL.g_areVBoundaries[RandomBoundary] + PMPS_GVL.reVHyst - PMPS_GVL.reVHyst/2,
         LastWord);
    TestEV := 0;
    TestEV.RandomBoundary := TRUE;
    TestEV.MNU := True;

    fbStr.arg1 := F_DWORD(Result);
    fbStr.arg2 := F_DWORD(TestEV);
    fbStr.sFormat := 'Moving up does not stick. Result: %b vs. Test: %b';
    fbStr();

AssertTrue(Result = TestEV,
    fbStr.sOut);

    Result := F_eVRangeCalculator(
        PMPS_GVL.g_areVBoundaries[RandomBoundary - 1] - PMPS_GVL.reVHyst + PMPS_GVL.reVHyst/2,
        LastWord);
    TestEV := 0;
    TestEV.RandomBoundary := TRUE;
    TestEV.MND := True;

    fbStr.arg1 := F_DWORD(Result);
    fbStr.arg2 := F_DWORD(TestEV);
    fbStr.sFormat := 'Moving down does not stick. Result: %b vs. Test: %b';
    fbStr();

AssertTrue(Result = TestEV,
    fbStr.sOut);

TEST_FINISHED();

Test('Check hyst drops');

    Result := F_eVRangeCalculator(
        PMPS_GVL.g_areVBoundaries[MND] - PMPS_GVL.reVHyst*1.1,
        LastWord);
    TestEV := 0;
    TestEV.MND := TRUE;

    fbStr.arg1 := F_DWORD(Result);
    fbStr.arg2 := F_DWORD(TestEV);
    fbStr.sFormat := 'Moving down does not drop. Result: %b vs. Test: %b';
    fbStr();

AssertTrue(Result = TestEV,
    fbStr.sOut);

    Result := F_eVRangeCalculator(
        PMPS_GVL.g_areVBoundaries[RandomBoundary] + PMPS_GVL.reVHyst*1.1,
        LastWord);
    TestEV := 0;
    TestEV.MNU := TRUE;

    fbStr.arg1 := F_DWORD(Result);
    fbStr.arg2 := F_DWORD(TestEV);
    fbStr.sFormat := 'Moving up does not drop. Result: %b vs. Test: %b';
    fbStr();

AssertTrue(Result = TestEV,
    fbStr.sOut);

TEST_FINISHED();
END_METHOD

END_FUNCTION_BLOCK

// TestComponents/FB_eVWithinSpec_Test
{attribute 'call_after_init'}
FUNCTION_BLOCK FB_eVWithinSpec_Test EXTENDS TcUnit.FB_TestSuite
VAR_INPUT
END_VAR
VAR_OUTPUT
END_VAR
VAR
END_VAR

evWithinRangeChecks();

METHOD evWithinRangeChecks
VAR_INPUT
END_VAR
VAR

END_VAR
TEST('evWithinRangeChecks');

//Upper limit equal
AssertTrue(
    F_eVWithinSpec(300, 2#0000_0000_0000_0010),
    'Upper limit not inclusive');
//Lower limit equal
AssertTrue(
    F_eVWithinSpec(300, 2#0000_0000_0000_0100),
    'Lower limit not inclusive');
//Out of range
AssertFalse(
    F_eVWithinSpec(300.1, 2#0000_0000_0000_0010),
    'Out of range failed, whatever you did, it broke this really bad.');
//Negative eV
AssertFalse(
    F_eVWithinSpec(-300, 16#FFFF),
    'Working with antimatter? Negative eV should not be acceptable.');
//Upper unallocated range
AssertFalse(
    F_eVWithinSpec(1701, 2#1000_0000_0000_0000),
    'eV range should not evaluate past 1.7keV');

TEST_FINISHED();
END_METHOD

END_FUNCTION_BLOCK

// TestComponents/FB_FastFault_Test
{attribute 'call_after_init'}
{attribute 'no_check'}
FUNCTION_BLOCK FB_FastFault_Test EXTENDS TcUnit.FB_TestSuite
VAR_INPUT
END_VAR
VAR_OUTPUT
END_VAR
VAR
    fbTime : FB_LocalSystemTime := ( bEnable := TRUE, dwCycle := 1 ); //Get current system time, used for override
END_VAR
VAR CONSTANT
    OvrdTime : TIME := T#2s;
END_VAR

FFCombinedFunctionality();
FFRegistration();
FFOvrdAndNextFault();

METHOD FFCombinedFunctionality
VAR_INPUT
END_VAR
VAR_INST
    fbFF    :    FB_FastFault;
    fbFFO    :    FB_HardwareFFOutput;

END_VAR
TEST('FFCombinedFunctionality');

//Clear initial faults
fbFFO.i_xReset:=TRUE; //Reset requested at start of cycle

fbFF(io_fbFFHWO := fbFFO, //FF reset somehwere in code
    i_xOK := TRUE,
    i_xReset := TRUE);

fbFFO.EvaluateOutput(); //FFO eval called at end of cycle

AssertTrue(fbFFO.q_xFastFaultOut,
    'Fast fault did not clear');


//Induce fault with FF

fbFFO(i_xReset := FALSE); //Reset released at start of cycle

fbFF(io_fbFFHWO := fbFFO, //FF faulted
    i_xOK := FALSE); //Reset is still set true from last call.

fbFFO.EvaluateOutput(); //FFO eval called at end of cycle

AssertFalse(fbFFO.q_xFastFaultOut,
    'Fast fault did not trip the beam');


//FFO remains faulted until local (FF) and FFO receieve fresh reset request, and faults
//are actually cleared

//Attempt to clear FFO fails because FF still faulted
fbFFO.i_xReset := TRUE; //Reset requested

fbFF(io_fbFFHWO := fbFFO, //FF faulted
    i_xOK := FALSE,
    i_xReset := FALSE);

fbFFO.EvaluateOutput(); //FFO eval called at end of cycle

AssertFalse(fbFFO.q_xFastFaultOut,
    'Fast fault output cleared while fault remains, very bad');

//Attempt to clear FF while fault remains fails
fbFFO.EvaluateOutput(i_xReset := FALSE);

fbFFO.i_xReset := TRUE; //Reset requested

fbFF(io_fbFFHWO := fbFFO, //FF faulted
    i_xOK := FALSE,
    i_xReset := TRUE); //This reset should fail.

fbFFO.EvaluateOutput(); //FFO eval called at end of cycle

AssertFalse(fbFFO.q_xFastFaultOut,
    'Fast fault cleared while fault remains, very bad');

TEST_FINISHED();
END_METHOD

{attribute 'no_check'}
METHOD FFOvrdAndNextFault
VAR_INPUT
END_VAR
VAR_INST
    fbFF    :    FB_FastFault :=(
        i_xAutoReset := TRUE);
    fbFFO    :    FB_HardwareFFOutput := (i_sNetID:='',
        bAutoReset := TRUE);
    rFF : REFERENCE TO ST_FF;

    FirstPass : BOOL := TRUE;
    fbTimePass : BOOL := TRUE;
    OvrdActvTstDone : BOOL := FALSE;

    TestsDone : BOOL := FALSE;
    Now: DATE_AND_TIME;
    Expiration : DINT;
    OvdTime : TIME ;
    Expire: TIMESTRUCT;
//seconds:ULINT;
    specificLocalTimeToFileTime : FB_TzSpecificLocalTimeToFileTime;
    fileTime: T_FILETIME;
END_VAR
TEST('FFVetoAndNextFault');
fbTime();

// I noticed something weird going on with the PEWatcher on the L line. It was faulted, and the fast fault
// was not tripping off beam. It had been previously overridden so I was wondering why it wasn't causing a trip.

IF  FirstPass  THEN

    fbFF(io_fbFFHWO := fbFFO, //FF reset somehwere in code
        i_xOK := TRUE);

    fbFFO.ExecuteNoLog(); //FFO eval called at end of cycle

    AssertTrue(fbFFO.q_xFastFaultOut,
        'Fast fault did not clear');


    //Induce fault with FF

    fbFF(io_fbFFHWO := fbFFO, //FF faulted
        i_xOK := FALSE);

    fbFFO.ExecuteNoLog(); //FFO eval called at end of cycle

    AssertFalse(fbFFO.q_xFastFaultOut,
        'Fast fault did not trip the beam');

    rFF REF= fbFFO.astFF[fbFF.RegistrationIdx];

FirstPass := FALSE;

END_IF


IF fbTime.bValid AND fbTimePass  THEN

    Now := SystemTime_TO_DT(fbTime.systemTime);
    Expire:= fbTime.systemTime;
    Expire.wSecond:= Expire.wSecond+5;
    specificLocalTimeToFileTime(in := Tc2_Utilities.SYSTEMTIME_TO_FILETIME(Expire), tzInfo := , out => fileTime);
    Expiration := TO_DINT((SHL(DWORD_TO_ULINT(fileTime.dwHighDateTime), 32) + DWORD_TO_ULINT(fileTime.dwLowDateTime)) / 10000000 - 11644473600);;

    WRITE_PROTECTED_DINT(ADR(rFF.Ovrd.Expiration), Expiration );
    WRITE_PROTECTED_TIME(ADR(rFF.Ovrd.Timer.PT), OvrdTime );
    WRITE_PROTECTED_BOOL(ADR(rFF.Ovrd.Activate), TRUE);

    fbTimePass:=FALSE;

END_IF

// On every cycle:
fbFF(io_fbFFHWO := fbFFO, //FF faulted
    i_xOK := FALSE);

fbFFO.ExecuteNoLog(); //FFO eval called at end of cycle


IF rFF.Ovrd.Active AND rFF.BeamPermitted THEN

    AssertTrue(fbFFO.q_xFastFaultOut,
        'Fast fault should be overridden so FFO should be true');

    OvrdActvTstDone := TRUE;
END_IF

IF OvrdActvTstDone and NOT rFF.Ovrd.Active and not rff.BeamPermitted THEN

    AssertFalse(fbFFO.q_xFastFaultOut,
        'Fast fault override expired so beam should be off.');
   // AssertFalse(rFF.BeamPermitted, 'Beam should not be permitted now');

    TestsDone := TRUE;
END_IF


IF TestsDone THEN
    TEST_FINISHED_NAMED('FFVetoAndNextFault');
END_IF
END_METHOD

{attribute 'no_check'}
METHOD FFRegistration
VAR_INPUT
END_VAR
VAR_INST
    fbFF    :    FB_FastFault;
    fbFFO    :    FB_HardwareFFOutput;
    astFF : ARRAY[0..10] OF ST_FF;
END_VAR
TEST('FFRegistration');

fbFF(io_fbFFHWO := fbFFO);

AssertEquals_STRING(fbFF.sPath, fbFFO.astFF[fbFF.RegistrationIdx].Info.sPath,
    'FF registration with FFO did not succeed');

TEST_FINISHED();
END_METHOD

END_FUNCTION_BLOCK

// TestComponents/FB_PhotonEnergyWatcher_Test
{attribute 'call_after_init'}
FUNCTION_BLOCK FB_PhotonEnergyWatcher_Test EXTENDS TcUnit.FB_TestSuite
VAR_INPUT
END_VAR
VAR_OUTPUT
END_VAR
VAR

END_VAR

PEWatcherBasicFunction();

METHOD PEWatcherBasicFunction
VAR_INPUT
END_VAR
VAR_INST
    fbPEW    :    FB_PhotonEnergyWatcher;
    fbFFO    :    FB_HardwareFFOutput;
    q_Output    :    BOOL;

    stCurBeamParams    :    ST_BeamParams;
    stMachineTargetBeamParams    :    ST_BeamParams;
    stReqBeamParams    :    ST_BeamParams;
END_VAR
TEST('PEWatcherBasicFunction');

//Clear FFO fault to start
fbFFO(i_xReset:=TRUE);

//All eV OK
stCurBeamParams.neVRange := F_eVRangeCalculator(800, 0);

stMachineTargetBeamParams.neVRange := 2#0000_0000_1000_0000;

stReqBeamParams.neVRange := 2#1111_1111_1111_1111;

fbFFO(i_xReset:=FALSE); //Reset request released

fbPEW(i_stCurrentBeamParams := stCurBeamParams,
    i_stMachineTargetBeamParams := stMachineTargetBeamParams,
    i_stRequestedBeamParams := stReqBeamParams,
    io_fbFFHWO := fbFFO,
    i_xReset := TRUE); //Clear local FF within PEW

fbFFO.EvaluateOutput(q_xFastFaultOut=>q_Output); //This simulates a completed PLC cycle
//Evaluate output should be called once at the end of a PLC cycle.

AssertTrue(q_Output,
    'Beam within limits, FFO should be true');


//Req eV moved out of range
stCurBeamParams.neVRange := F_eVRangeCalculator(800, 0);

stMachineTargetBeamParams.neVRange := F_eVRangeCalculator(800, 0);

stReqBeamParams.neVRange := 2#0000_1111_0011_1111;

fbPEW.i_xReset := FALSE; //release local FF reset req
fbPEW(i_stCurrentBeamParams := stCurBeamParams,
    i_stMachineTargetBeamParams := stMachineTargetBeamParams,
    i_stRequestedBeamParams := stReqBeamParams,
    io_fbFFHWO := fbFFO);

fbFFO.EvaluateOutput(q_xFastFaultOut=>q_Output);

AssertFalse(q_Output,
    'Limits moved beyond current and target beam, should produce a fault.');

//Beam and target eV moved back within permitted ranges, reset clears fault
stCurBeamParams.neVRange := F_eVRangeCalculator( 300, 0);

stMachineTargetBeamParams.neVRange := F_eVRangeCalculator(300, 0);

stReqBeamParams.neVRange := 2#0000_1111_0011_1111;

fbFFO(i_xReset:=TRUE); //New reset request

fbPEW.i_xReset := TRUE; //New reset request

fbPEW(i_stCurrentBeamParams := stCurBeamParams, //Beam params are now within spec
    i_stMachineTargetBeamParams := stMachineTargetBeamParams,
    i_stRequestedBeamParams := stReqBeamParams,
    io_fbFFHWO := fbFFO);

fbFFO.EvaluateOutput(q_xFastFaultOut=>q_Output);

AssertTrue(q_Output,
    'Beam within limits after reset, FFO should be true');

//At this point, the fast fault would be cleared

//Current beam eV moved out of range
stCurBeamParams.neVRange := F_eVRangeCalculator(800, 0); //Moved out of range

stMachineTargetBeamParams.neVRange := F_eVRangeCalculator(300, 0); //Still within range

stReqBeamParams.neVRange := 2#0000_1111_0011_1111;

fbPEW(i_stCurrentBeamParams := stCurBeamParams,
    i_stMachineTargetBeamParams := stMachineTargetBeamParams,
    i_stRequestedBeamParams := stReqBeamParams,
    io_fbFFHWO := fbFFO);

fbFFO.EvaluateOutput(q_xFastFaultOut=>q_Output);

AssertFalse(q_Output,
    'Current beam moved beyond set limits, should produce a fault');

//Target beam eV moved out of range
fbFFO(i_xReset:=FALSE); //Reset released
fbFFO(i_xReset:=TRUE); //New reset request comes in at the top of a cycle, but will be overridden

stCurBeamParams.neVRange := F_eVRangeCalculator(300, 0); //Now within range

stMachineTargetBeamParams.neVRange := F_eVRangeCalculator(800, 0); //Moved out of range

stReqBeamParams.neVRange := 2#0000_1111_0011_1111;

fbPEW.i_xReset := TRUE; //Attempt to reset local FF will fail
fbPEW(i_stCurrentBeamParams := stCurBeamParams,
    i_stMachineTargetBeamParams := stMachineTargetBeamParams,
    i_stRequestedBeamParams := stReqBeamParams,
    io_fbFFHWO := fbFFO);

fbFFO.EvaluateOutput(q_xFastFaultOut=>q_Output);

AssertFalse(q_Output,
    'Target beam moved beyond set limits, should produce a fault');

TEST_FINISHED();
END_METHOD

END_FUNCTION_BLOCK

// TestComponents/FB_SafeBPCompare_Test
{attribute 'call_after_init'}
FUNCTION_BLOCK FB_SafeBPCompare_Test EXTENDS TcUnit.FB_TestSuite
VAR_INPUT
END_VAR
VAR_OUTPUT
END_VAR
VAR

END_VAR

BeamOffIsSafe();
BPComparisonCheck();

//Verify beam off is considered safe.
METHOD BeamOffIsSafe
VAR_INPUT
END_VAR
VAR
    stBeamOn_MoreConservative    :    ST_BeamParams;
    stBeamOff_LessConservative    :    ST_BeamParams;
    stBeam0Rate    :    ST_BeamParams;
    stBeam0BC    :    ST_BeamParams;
    fb_BeamClassOutputs_BCD:FB_BeamClassOutputs_BCD;
END_VAR
stBeamOn_MoreConservative  := F_SetBeamParams(
    0, //0% transmission is more conservative than 50
    16#FFFF_FFFF,
    120, //rate
    16#0001,
    PMPS_GVL.DUMMY_AUX_ATT_ARRAY);

stBeamOff_LessConservative:= F_SetBeamParams(
    0.5, //50% transmission, less conservative, without 0-rate this beam parameter set would be less safe than above
    16#FFFF_FFFF,
    0, //rate, hence, more conservative
    16#000F,
    PMPS_GVL.DUMMY_AUX_ATT_ARRAY); //0 beam rate means this bps is actually safer than BeamOn

// Set Machine Mode to NC
PMPS_GVL.stCurrentBeamParameters.nMachineMode := 0;

TEST('BeamOffIsSafeNC');

AssertTrue(
    F_SafeBPCompare0Rate(stBeamOff_LessConservative, stBeamOn_MoreConservative),
    'SafeBPCompare in NC does not think beam rate = 0 is safer than anything else.');
TEST_FINISHED();


TEST('BeamClass0IsNOTSafeNC');


stBeam0BC  := F_SetBeamParams(
    1, //0% transmission is more conservative than 50
    16#FFFF_FFFF,
    1000, //rate
    16#0000,
    PMPS_GVL.DUMMY_AUX_ATT_ARRAY);


AssertFalse(
    F_SafeBPCompare0Rate(stBeam0BC, stBeamOn_MoreConservative),
    'SafeBPCompare beam class = 0 is NOT safer than anything else in NC mode.');
TEST_FINISHED();




//SC tests
stBeamOn_MoreConservative  := F_SetBeamParams(
    0, //0% transmission is more conservative than 50
    16#FFFF_FFFF,
    0, //rate
    16#000F,
    PMPS_GVL.DUMMY_AUX_ATT_ARRAY);

stBeamOff_LessConservative:= F_SetBeamParams(
    0.5, //50% transmission, less conservative, without 0-rate this beam parameter set would be less safe than above
    16#FFFF_FFFF,
    1000,
    16#0000, //zero beam, hence, more conservative
    PMPS_GVL.DUMMY_AUX_ATT_ARRAY); //0 beam rate means this bps is actually safer than BeamOn

// Set Machine Mode to SC
PMPS_GVL.stCurrentBeamParameters.nMachineMode := 1;

TEST('BeamOffIsSafeSC');

AssertTrue(
    F_SafeBPCompare0Rate(stBeamOff_LessConservative, stBeamOn_MoreConservative),
    'SafeBPCompare in SC mode does not think beam class = 0 is safer than anything else.');
TEST_FINISHED();

TEST('Beam0RateIsNOTSafeSC');


stBeam0Rate  := F_SetBeamParams(
    1, //0% transmission is more conservative than 50
    16#FFFF_FFFF,
    0, //rate
    16#00FF,
    PMPS_GVL.DUMMY_AUX_ATT_ARRAY);


AssertFalse(
    F_SafeBPCompare0Rate(stBeam0Rate, stBeamOn_MoreConservative),
    'SafeBPCompare beam rate = 0 is NOT safer than anything else in SC mode.');
TEST_FINISHED();


// Set Machine Mode to Misconfigured
PMPS_GVL.stCurrentBeamParameters.nMachineMode := 2;
TEST('WrongMachineMode');

AssertFalse(
    F_SafeBPCompare0Rate(stBeam0Rate, stBeam0BC),
    'SafeBPCompare in Misconfigured mode does not think beam rate = 0 is safer than anything else.');

AssertFalse(
    F_SafeBPCompare0Rate(stBeam0BC, stBeam0Rate),
    'SafeBPCompare in Misconfiigured mode does not think beam class = 0 is safer than anything else.');
TEST_FINISHED();
END_METHOD

//Verify BP comparison remains logical.
{attribute 'no_check'}
METHOD BPComparisonCheck
VAR_INPUT
END_VAR
VAR
    stSafer    :    ST_BeamParams;
    stNotSoSafe    :    ST_BeamParams;
    idx : UINT;

    xResult : BOOL;
    xFailedTest : BOOL; // To exit loops early
END_VAR
// Test in NC mode
PMPS_GVL.stCurrentBeamParameters.nMachineMode :=0;

TEST('BPComparisonTran');
//Attenuation
stSafer := F_SetBeamParams(
    0.51, //
    16#FFFFFFFF,
    1,
    16#0000,
    PMPS_GVL.DUMMY_AUX_ATT_ARRAY);

stNotSoSafe := F_SetBeamParams(
    0.62, //
    16#FFFFFFFF,
    1,
    16#0000,
    PMPS_GVL.DUMMY_AUX_ATT_ARRAY);

AssertTrue(
    F_SafeBPCompare(stSafer, stNotSoSafe),
    'Attenuation eval is broken (True)');

AssertFalse(
    F_SafeBPCompare(stNotSoSafe, stSafer),
    'Attenuation eval is broken (False)');

// Check at margin threshold
stSafer.nTran := 0.99 * stNotSoSafe.nTran*(PMPS_GVL.TRANS_SCALING_FACTOR + PMPS_PARAM.TRANS_MARGIN)/PMPS_GVL.TRANS_SCALING_FACTOR;
AssertTrue(
    F_SafeBPCompare(stSafer, stNotSoSafe),
    'Attenuation eval is broken: should be safe up to margin.');

stSafer.nTran := 1 + stNotSoSafe.nTran*(PMPS_GVL.TRANS_SCALING_FACTOR + PMPS_PARAM.TRANS_MARGIN)/PMPS_GVL.TRANS_SCALING_FACTOR;

AssertFalse(
    F_SafeBPCompare(stSafer, stNotSoSafe),
    'Attenuation eval is broken (False): should not be safe at all past margin');

TEST_FINISHED();



//Attenuator array
TEST('BPComparisonTranArray');

stSafer := F_SetBeamParams(
    0, //
    16#FFFFFFFF,
    1,
    16#0000,
    PMPS_GVL.DUMMY_AUX_ATT_ARRAY);

stNotSoSafe := F_SetBeamParams(
    0, //
    16#FFFFFFFF,
    1,
    16#000F,
    PMPS_GVL.DUMMY_AUX_ATT_ARRAY);

FOR idx:=1 TO PMPS_GVL.AUX_ATTENUATORS DO
    stSafer.astAttenuators[idx].nTran := 0.00500;
    stNotSoSafe.astAttenuators[idx].nTran := 0.00600;

    xResult := F_SafeBPCompare(stSafer, stNotSoSafe);

    AssertTrue(
    xResult,
    'Attenuation array eval is broken (True)');

    xFailedTest S= NOT xResult;

    xResult := F_SafeBPCompare(stNotSoSafe, stSafer);
    AssertFalse(
    xResult,
    'Attenuation array eval is broken (False)');

    xFailedTest S= xResult;

    // Check at margin threshold
        stSafer.astAttenuators[idx].nTran := stNotSoSafe.astAttenuators[idx].nTran*(PMPS_GVL.TRANS_SCALING_FACTOR + PMPS_PARAM.TRANS_MARGIN)/PMPS_GVL.TRANS_SCALING_FACTOR;

        xResult := F_SafeBPCompare(stSafer, stNotSoSafe);

        AssertTrue(
            xResult,
            'Attenuation eval is broken: should be safe up to margin.');
        xFailedTest S= NOT xResult;

        stSafer.astAttenuators[idx].nTran := 1 + stNotSoSafe.astAttenuators[idx].nTran*(PMPS_GVL.TRANS_SCALING_FACTOR + PMPS_PARAM.TRANS_MARGIN)/PMPS_GVL.TRANS_SCALING_FACTOR;

        xResult := F_SafeBPCompare(stSafer, stNotSoSafe);
        AssertFalse(
            xResult,
            'Attenuation eval is broken (False): should not be safe at all past margin');
        xFailedTest S= xResult;
    //////////////////////
    IF xFailedTest THEN
        stSafer.astAttenuators[idx].nTran := 0;
        stNotSoSafe.astAttenuators[idx].nTran := 0;
        xFailedTest := FALSE;
        EXIT; // Exit this loop on the first failure.
    END_IF

    stSafer.astAttenuators[idx].nTran := 0;
    stNotSoSafe.astAttenuators[idx].nTran := 0;

END_FOR

TEST_FINISHED();

stSafer.astAttenuators[idx].nTran := 0;
stNotSoSafe.astAttenuators[idx].nTran := 0;

//Aperture array
TEST('BPComparisonApertureArray');

FOR idx:=1 TO PMPS_GVL.MAX_APERTURES DO
    // Height
    stSafer.astApertures[idx].Height := 30; // narrower is safer
    stNotSoSafe.astApertures[idx].Height := 50;

    AssertTrue(
    F_SafeBPCompare(stSafer, stNotSoSafe),
    'Aperture array eval is broken on height (True)');

    AssertFalse(
    F_SafeBPCompare(stNotSoSafe, stSafer),
    'Aperture array eval is broken on height (False)');

    IF NOT F_SafeBPCompare(stSafer, stNotSoSafe) or F_SafeBPCompare(stNotSoSafe, stSafer) THEN
        EXIT; // Exit this loop on the first failure.
    END_IF

    stSafer.astApertures[idx].Height := 0;
    stNotSoSafe.astApertures[idx].Height := 0;

    // Width
    stSafer.astApertures[idx].Width := 30; // narrower is safer
    stNotSoSafe.astApertures[idx].Width := 50;

    AssertTrue(
    F_SafeBPCompare(stSafer, stNotSoSafe),
    'Aperture array eval is broken on width (True)');

    AssertFalse(
    F_SafeBPCompare(stNotSoSafe, stSafer),
    'Aperture array eval is broken on width (False)');

    IF NOT F_SafeBPCompare(stSafer, stNotSoSafe) or F_SafeBPCompare(stNotSoSafe, stSafer) THEN
        EXIT; // Exit this loop on the first failure.
    END_IF

    stSafer.astApertures[idx].Width := 0;
    stNotSoSafe.astApertures[idx].Width := 0;


END_FOR

TEST_FINISHED();

//Rate
TEST('BPComparisonRate');
stSafer := F_SetBeamParams(
    0,
    16#FFFF_FFFF,
    1,
    16#0000,
    PMPS_GVL.DUMMY_AUX_ATT_ARRAY); //

stNotSoSafe := F_SetBeamParams(
    0,
    16#FFFF_FFFF,
    10,
    16#0001,
    PMPS_GVL.DUMMY_AUX_ATT_ARRAY); //

AssertTrue(
    F_SafeBPCompare(stSafer, stNotSoSafe),
    'Rate eval is broken (True)');

AssertFalse(
    F_SafeBPCompare(stNotSoSafe, stSafer),
    'Rate eval is broken (False)');
TEST_FINISHED();

//Pulse energy
(*
TEST('BPComparisonPulseEnergy');
stSafer := F_SetBeamParams(
    0,
    1, //
    16#FFFF,
    1,
    PMPS_GVL.DUMMY_AUX_ATT_ARRAY);

stNotSoSafe := F_SetBeamParams(
    0,
    10, //
    16#FFFF,
    1,
    PMPS_GVL.DUMMY_AUX_ATT_ARRAY);
    *)
AssertTrue(
    F_SafeBPCompare(stSafer, stNotSoSafe),
    'Pulse energy eval is broken (True)');

AssertFalse(
    F_SafeBPCompare(stNotSoSafe, stSafer),
    'Pulse energy eval is broken (False)');
TEST_FINISHED();

//Photon energy
//More extensive tests elsewhere
TEST('BPComparisonPhotonEnergy');
stSafer := F_SetBeamParams(
    0,
    2#0000_0000_0000_0000_0000_0000_0000_0010,
    1,
    16#0000,
    PMPS_GVL.DUMMY_AUX_ATT_ARRAY);

stNotSoSafe := F_SetBeamParams(
    0,
    2#0000_0000_0000_0000_0000_0000_0000_0110,
    1,
    16#0001,
    PMPS_GVL.DUMMY_AUX_ATT_ARRAY);

AssertTrue(
    F_SafeBPCompare(stSafer, stNotSoSafe),
    'Photon energy eval is broken (True)');

AssertFalse(
    F_SafeBPCompare(stNotSoSafe, stSafer),
    'Photon energy eval is broken (False)');
TEST_FINISHED();
END_METHOD

END_FUNCTION_BLOCK

// TestComponents/FB_SubsysToArb_Test
{attribute 'call_after_init'}
FUNCTION_BLOCK FB_SubsysToArb_Test EXTENDS TcUnit.FB_TestSuite
VAR_INPUT
END_VAR
VAR_OUTPUT
END_VAR
VAR
END_VAR

BasicFunction();
VetoFunction();

{attribute 'no_check'}
METHOD BasicFunction
VAR_INPUT
END_VAR
VAR
    nId    :    DWORD := 1;
    stReq    :    ST_BeamParams := (nTran:=12);
END_VAR
VAR_INST
    fbArbiter    :    FB_Arbiter(1);

    fbSubSysToArb : FB_SubSysToArbiter_IO; // Subsystem interface with beamline arbiter PLC
    pBPC : POINTER TO ST_BeamParams_IO;

    ioCurrentBP : ST_BeamParams_IO;

    FFO : FB_HardwareFFOutput; // Dummy FFO not important for these tests

    nCohortScratch : UDINT;

END_VAR
VAR CONSTANT
    SysID : DWORD := 42;
END_VAR
// This simulates a synchronous cycle between the subsystem and arbiter PLC cycles. Ie. phase is locked, and cycle time is the same. This is not always the case, so these tests should be
// trusted with a grain of salt.

TEST('Add to arbiter');

IF NOT fbArbiter.CheckRequestInPool(nID) THEN
    AssertTrue(fbArbiter.AddRequest(nId, stReq,'Device'), 'Arbiter returned false from AddRequest'); // some device asking its local arbiter for some beam parameters
END_IF

TEST_FINISHED();

///////////////////////////////////////
//Sub system cycle
fbSubSysToArb(Arbiter := fbArbiter, fbFFHWO := FFO);
//END of sub system cycle
///////////////////////////////////////


TEST('Initial Elevation');
AssertTrue(fbSubSysToArb.nRequestCohort = fbSubSysToArb.q_stRequestedBP.nCohortInt, 'ReqCohort and qBP Cohort do not match');
AssertFalse(fbArbiter.nActiveCohort <> 0, 'Arbiter indicates it is included in arbitration prematurely');
AssertTrue(fbSubSysToArb.nRequestCohort <> 0, 'Cohort index should move to 1 with first request');
TEST_FINISHED_NAMED('Initial Elevation');

nCohortScratch := fbSubSysToArb.nRequestCohort;

//Ethercat transfer simulation
// Transfer of requested BP to arbiter PLC
// pBPR := ADR(fbArbToSubSys.i_RequestedBP);
// pBPR^ := fbSubSysToArb.q_stRequestedBP;

ioCurrentBP := fbSubSysToArb.q_stRequestedBP;
// NOTE: Setting the returning cohort number to something less than the request cohort number
// will prevent the sub system arbiter FB from considering itself active in arbitration.
// The next set of tests verify this.
ioCurrentBP.nCohortInt := 0;

// Transfer of current BP to sub system PLC
pBPC := ADR(fbSubSysToArb.i_stCurrentBP);
pBPC^ := ioCurrentBP;

///////////////////////////////////////
//Sub system cycle
fbSubSysToArb(Arbiter := fbArbiter, fbFFHWO := FFO);
//END of sub system cycle
///////////////////////////////////////

TEST('Not yet active in arbitration');
AssertTrue(fbSubSysToArb.nActiveCohort = 0, 'Active cohort should still be zero, per ioCurrentBP.nCohortInt setting above.');
AssertFalse(fbArbiter.nActiveCohort <> 0, 'Arbiter indicates it is included in arbitration prematurely, checkrequest might be broken');
AssertTrue(fbSubSysToArb.nRequestCohort = nCohortScratch, 'Cohort index should not have changed because there have been no additional requests added to the arbiter');
TEST_FINISHED_NAMED('Not yet active in arbitration');

//Ethercat transfer simulation
// Transfer of requested BP to arbiter PLC
// pBPR := ADR(fbArbToSubSys.i_RequestedBP);
// pBPR^ := fbSubSysToArb.q_stRequestedBP;

ioCurrentBP := fbSubSysToArb.q_stRequestedBP;
// NOTE: Now we simulate the FB_ArbiterToSubSys_IO updating the cohort number to the same value as the request cohort, indicating that cohort has been included
ioCurrentBP.nCohortInt := 2;

// Transfer of current BP to sub system PLC
pBPC := ADR(fbSubSysToArb.i_stCurrentBP);
pBPC^ := ioCurrentBP;

///////////////////////////////////////
//Sub system cycle
fbSubSysToArb(Arbiter := fbArbiter, fbFFHWO := FFO);
//END of sub system cycle
///////////////////////////////////////

TEST('Active in arbitration');
AssertTrue(fbSubSysToArb.nActiveCohort = fbSubSysToArb.nRequestCohort, 'Active cohort and request cohort do not match');
AssertTrue(fbArbiter.nActiveCohort = 1, 'Arbiter does not indicate it is included in higher arbitration');
TEST_FINISHED_NAMED('Active in arbitration');
END_METHOD

METHOD VetoFunction
VAR_INPUT
END_VAR
VAR
    nId    :    DWORD := 1;
    stReq    :    ST_BeamParams := (nTran:=12);
END_VAR
VAR_INST
    fbArbiter    :    FB_Arbiter(1);

    fbSubSysToArb : FB_SubSysToArbiter_IO; // Subsystem interface with beamline arbiter PLC
    fbArbToSubSys : FB_ArbiterToSubSys_IO;

    pBPC : POINTER TO ST_BeamParams_IO;
    pBPR : POINTER TO ST_BeamParams_IO;

    ioCurrentBP : ST_BeamParams_IO;

    FFO : FB_HardwareFFOutput; // Dummy FFO not important for these tests

END_VAR
VAR CONSTANT
    SysID : DWORD := 42;
END_VAR
// This simulates a synchronous cycle between the subsystem and arbiter PLC cycles. Ie. phase is locked, and cycle time is the same. This is not always the case, so these tests should be
// trusted with a grain of salt.

fbArbiter.AddRequest(nId, stReq,'Device'); // some device asking its local arbiter for some beam parameters


///////////////////////////////////////
//Sub system cycle
fbSubSysToArb(Arbiter := fbArbiter, fbFFHWO := FFO);
//END of sub system cycle
///////////////////////////////////////

TEST('Request propagated');
    AssertTrue(fbSubSysToArb.q_stRequestedBP.nTran = stReq.nTran, 'Request not propagated');
TEST_FINISHED();

// Veto activated
///////////////////////////////////////
//Sub system cycle
fbSubSysToArb(Arbiter := fbArbiter, fbFFHWO := FFO, i_bVeto:=TRUE);
//END of sub system cycle
///////////////////////////////////////

// Veto activated
///////////////////////////////////////
//Sub system cycle
fbSubSysToArb(Arbiter := fbArbiter, fbFFHWO := FFO, i_bVeto:=TRUE);
//END of sub system cycle
///////////////////////////////////////

TEST('Request sustained');
    AssertTrue(fbSubSysToArb.q_stRequestedBP.nTran = PMPS_GVL.cstFullBeam.nTran, 'Request still being propagated');
    AssertTrue(fbArbiter.CheckRequest(nId), 'Request still not valid');
TEST_FINISHED();

// Veto activated
///////////////////////////////////////
//Sub system cycle
fbSubSysToArb(Arbiter := fbArbiter, fbFFHWO := FFO, i_bVeto:=FALSE);
//END of sub system cycle
///////////////////////////////////////

// Veto activated
///////////////////////////////////////
//Sub system cycle
fbSubSysToArb(Arbiter := fbArbiter, fbFFHWO := FFO, i_bVeto:=FALSE);
fbSubSysToArb(Arbiter := fbArbiter, fbFFHWO := FFO, i_bVeto:=FALSE);
fbSubSysToArb(Arbiter := fbArbiter, fbFFHWO := FFO, i_bVeto:=FALSE);
//END of sub system cycle
///////////////////////////////////////

TEST('Request restored');
    AssertTrue(fbSubSysToArb.q_stRequestedBP.nTran = stReq.nTran, 'Request still being sustained');
TEST_FINISHED();
END_METHOD

END_FUNCTION_BLOCK

// TestComponents/FB_VetoArbiter_Test
{attribute 'call_after_init'}
FUNCTION_BLOCK FB_VetoArbiter_Test EXTENDS TcUnit.FB_TestSuite
VAR_INPUT
END_VAR
VAR_OUTPUT
END_VAR
VAR
END_VAR
VAR CONSTANT
    ArbID : DWORD := 1;
    HigherArbID : DWORD := 2;
END_VAR

VetoArbiter();

METHOD VetoArbiter

VAR_INPUT
END_VAR
VAR
    nId    :    DWORD := 1;
    nId2 : DWORD := 10;
    stReq    :  ST_BeamParams := (nTran:=0.12);
    stReq2	:	ST_BeamParams := (nTran:=0.10);
END_VAR
VAR_INST
    fbArbiter    :    FB_Arbiter(1);

    fbHigherArb : FB_Arbiter(2);

    ArbBP : ST_BeamParams:=(nTran:=1);

    VetoArb : FB_VetoArbiter;

    FFO : FB_HardwareFFOutput;

    fbHA : FB_DummyHA;

END_VAR

TEST('VetoNotIn');
fbArbiter.AddRequest(nReqID:=nId, stReqBP:=stReq, sDevName :='Device');

//////////////////// Cycle
fbHigherArb.ElevateRequest(fbHA);

VetoArb.bVeto := FALSE;
VetoArb(HigherAuthority:=fbHigherArb,
    LowerAuthority:=fbArbiter,
    FFO:=FFO);

//////////////////// Cycle
fbHigherArb.ElevateRequest(fbHA);

VetoArb.bVeto := FALSE;
VetoArb(HigherAuthority:=fbHigherArb,
    LowerAuthority:=fbArbiter,
    FFO:=FFO);

AssertTrue(fbHigherArb.q_stBeamParams.nTran = stReq.nTran, 'We should see the transmission number here, veto device is not in');

TEST_FINISHED();

TEST('VetoIn');
// Veto device is in
// This should effectively remove the fbArbiter request from the higher arbiter pool

//////////////////// Cycle
fbHigherArb.ElevateRequest(fbHA);

VetoArb.bVeto := TRUE;
VetoArb(HigherAuthority:=fbHigherArb, // Veto removed
    LowerAuthority:=fbArbiter,
    FFO:=FFO);

//////////////////// Cycle
fbHigherArb.ElevateRequest(fbHA);

VetoArb.bVeto := TRUE;
VetoArb(HigherAuthority:=fbHigherArb, // Veto removed
    LowerAuthority:=fbArbiter,
    FFO:=FFO);

AssertTrue(fbHigherArb.q_stBeamParams.nTran = PMPS_GVL.cstFullBeam.nTran, 'Veto device is in, trans should be restored to 100');
AssertTrue(fbArbiter.CheckRequest(nId), 'Request should still be considered valid (1)');
AssertFalse(fbHigherArb.CheckRequest(ArbID), 'Lower arb request should be gone from the higher pool');

TEST_FINISHED();

TEST('AnotherRequest');
// Another request is added, should be approved immediately, and with no effect on the final set
fbArbiter.RequestBP(nReqID := nId2, stReqBP:=stReq2);

//////////////////// Cycle
fbHigherArb.ElevateRequest(fbHA);

VetoArb.bVeto := TRUE;
VetoArb(HigherAuthority:=fbHigherArb, // Veto removed
    LowerAuthority:=fbArbiter,
    FFO:=FFO);

//////////////////// Cycle
fbHigherArb.ElevateRequest(fbHA);

VetoArb.bVeto := TRUE;
VetoArb(HigherAuthority:=fbHigherArb, // Veto removed
    LowerAuthority:=fbArbiter,
    FFO:=FFO);

AssertTrue(ArbBP.nTran = PMPS_GVL.cstFullBeam.nTran, 'Veto device remained in, trans should still be 100');
AssertTrue(fbArbiter.CheckRequest(nId), 'Request should still be considered valid (2)');
AssertTrue(fbArbiter.CheckRequest(nId2), '2nd Request should be considered valid');

TEST_FINISHED();

TEST('RemoveVeto');
// Removal of veto device, should produce a fault
//////////////////// Cycle
fbHigherArb.ElevateRequest(fbHA);

VetoArb.bVeto := FALSE;
VetoArb(HigherAuthority:=fbHigherArb, // Veto removed
    LowerAuthority:=fbArbiter,
    FFO:=FFO);

AssertFalse(VetoArb.ffKeepItSecretKeepItSafe.i_xOK, 'Should produce a fast fault at this point because the request is not yet back in the pool');

//////////////////// Cycle
fbHigherArb.ElevateRequest(fbHA);

VetoArb.bVeto := FALSE;
VetoArb(HigherAuthority:=fbHigherArb, // Veto removed
    LowerAuthority:=fbArbiter,
    FFO:=FFO);

//////////////////// Cycle
fbHigherArb.ElevateRequest(fbHA);

VetoArb.bVeto := FALSE;
VetoArb(HigherAuthority:=fbHigherArb, // Veto removed
    LowerAuthority:=fbArbiter,
    FFO:=FFO);

//////////////////// Cycle
fbHigherArb.ElevateRequest(fbHA);

VetoArb.bVeto := FALSE;
VetoArb(HigherAuthority:=fbHigherArb, // Veto removed
    LowerAuthority:=fbArbiter,
    FFO:=FFO);

AssertTrue(VetoArb.ffKeepItSecretKeepItSafe.i_xOK, 'Fault should be gone.');

TEST_FINISHED();
END_METHOD

END_FUNCTION_BLOCK

// MAIN
PROGRAM MAIN
VAR
    fbSetPERanges : PE_Ranges;

    fbDiffBPTest    :    FB_DiffBP_Test;
    fbBPTMTest    :    FB_BPTM_Test;
    fbSafeBPCompareTest    :    FB_SafeBPCompare_Test;
    ////fbevWithinSpecTest    :    FB_evWithinSpec_Test;---
    ////fbPEWTest    :    FB_PhotonEnergyWatcher_Test;---
    fbFFTest    :    FB_FastFault_Test;
    fbArbiterTest    :    FB_Arbiter_Test;
    fbVetoArbiterTest : FB_VetoArbiter_Test;
    fbevRangeCalcTest : FB_evRangeCalculator_Test;
    fbSubSysToArbTest : FB_SubsysToArb_Test;
    fbArbToSubSysTest : FB_ArbToSubsys_Test;
END_VAR

TcUnit.RUN();

END_PROGRAM
